// TIA Portal V19 export
TYPE "LEXCHANGETRAY_typeHandlingXyzEm_toConstraintRollerRecieve"
// stored: Access Published
   STRUCT
      feedback : "LEXCHANGETRAY_typeConstraintRollerEm_toHandlingXyzFeedback";
      req { S7_SetPoint := 'True'} : "LEXCHANGETRAY_typeConstraintRollerEm_toHandlingXyzReq";
   END_STRUCT;
END_TYPE
